// TIA Portal V19 export
TYPE "LEXCHANGETRAY_typeHandlingXyzEm_toPlasticRecieve"
// stored: Access Published
   STRUCT
      feedback : "LEXCHANGETRAY_typePlasticEm5_toHandlingXyzFeedback";
      req { S7_SetPoint := 'True'} : "LEXCHANGETRAY_typePlasticEm5_toHandlingXyzReq";
   END_STRUCT;
END_TYPE
